Staubli VAL3: Day22.dtx

num nResult
num nStart[2]
num nEyes
num nDice
num nPointsP1_virt
num nPointsP1_sum
num nPointsP2_virt
num nPointsP2_sum
string sInput
lists lResult
  [0]
    string sString
string sCommand
num nCoord_X
string sCoord_X
lists lResultCoord
  [0]
    string sString
string sCoord_Y
string sCoord_Z
num nRange
num nRangeX
num nRangeY
num nCoord_Y
num nRangeZ
num nCoord_Z
bool bGrid[1 1 1]
